TYPE U_CAM_STATE :
UNION
  stState             : ARRAY[1..MAX_AXIS] OF ST_CAM_STATE;

  byState   AT %i*    : ARRAY[1..MAX_AXIS] OF
                        ARRAY[1..SIZEOF(ST_CAM_STATE)] OF BYTE;
END_UNION
END_TYPE

(* stored: Version 1.1.0.1
   DUT U_CAM_STATE: Id {3f5377fa-a8b9-43af-854f-2b7fc8942fbd} *)
